Fanuc KAREL source: KB00028.KL

PROGRAM KB00028
%NOLOCKGROUP
%ENVIRONMENT UIF
VAR
  P1: INTEGER
  P2: STRING[80]
  P3: INTEGER
BEGIN
  P1 = 1
  P2 = 'A'
  P3 = 1
  CNC_DYN_DISE(P1, P2, P3)
END KB00028
